// TIA Portal V19 export
DATA_BLOCK "InstCallInterfaceSignals"   // DB29
{ DB_Accessible_From_OPC_UA := 'FALSE' }
FAMILY : Diag
VERSION : 1.0
// stored: DBAccessibleFromOPCUA false, DBAccessibleFromWebserver false, InstanceOfName CallInterfaceSignals, InstanceOfType FB
"CallInterfaceSignals"
   // VAR
   //    statReadValueHmi : Bool;
   //    statSelectSignalsHmi : USInt;
   //    statSelectSignalsOld { ExternalAccessible := 'False'; ExternalVisible := 'False'; ExternalWritable := 'False'} : USInt;
   //    statRisEdgeReadName { ExternalAccessible := 'False'; ExternalVisible := 'False'; ExternalWritable := 'False'} : Bool;
   //    statPosPulseReadName : Bool;
   //    statInterfaceSignalsHmi : Array[0..16] of "LAF_typeInterfaceSignalsHmi";
   //    instSignals1Left { S7_SetPoint := 'True'} : "LAF_InterfaceSignalsBool";
   //    instSignals1Right { ExternalAccessible := 'False'; ExternalVisible := 'False'; ExternalWritable := 'False'} : "LAF_InterfaceSignalsBool";
   //    instSignals2Left { ExternalAccessible := 'False'; ExternalVisible := 'False'; ExternalWritable := 'False'} : "LAF_InterfaceSignalsBool";
   //    instSignals2Right { ExternalAccessible := 'False'; ExternalVisible := 'False'; ExternalWritable := 'False'} : "LAF_InterfaceSignalsBool";
   //    instSignals3Left { ExternalAccessible := 'False'; ExternalVisible := 'False'; ExternalWritable := 'False'} : "LAF_InterfaceSignalsBool";
   //    instSignals3Right { ExternalAccessible := 'False'; ExternalVisible := 'False'; ExternalWritable := 'False'} : "LAF_InterfaceSignalsBool";
   //    instSignals4Left { ExternalAccessible := 'False'; ExternalVisible := 'False'; ExternalWritable := 'False'} : "LAF_InterfaceSignalsBool";
   //    instSignals4Right { ExternalAccessible := 'False'; ExternalVisible := 'False'; ExternalWritable := 'False'} : "LAF_InterfaceSignalsBool";
   //    instSignals5Left { ExternalAccessible := 'False'; ExternalVisible := 'False'; ExternalWritable := 'False'} : "LAF_InterfaceSignalsBool";
   //    instSignals5Right { ExternalAccessible := 'False'; ExternalVisible := 'False'; ExternalWritable := 'False'} : "LAF_InterfaceSignalsBool";
   // END_VAR
BEGIN
END_DATA_BLOCK
